// Mitsubishi GX Works2 project: WheelValveTurn   PLC: FX1N/FX1NC

// task Task_01 (event TRUE, interval 0, priority 31): POU_01

PROGRAM POU_01
OUT(X0, Y0);
OUT(X1, Y1);
OUT(X2, Y2);
OUT(X3, Y3);
OUT(X4, Y4);
OUT(X5, Y5);
OUT(X6, Y6);
END_PROGRAM
